FUNCTION_BLOCK fb_palletizeing
VAR_INPUT
END_VAR
VAR_OUTPUT
END_VAR
VAR
	SFCInit: BOOL;
	fbi_coordinateCal: fb_coordinateCal;
	fbi_exchangeTraySystem: fb_exchangeTraySystem;
	trn_pickUpLensDone: BOOL;
	trn_forTray: BOOL;
	trn_forGarbage: BOOL;
	trn_forSample: BOOL;
	trn_trayDone: BOOL;
	trn_garbageDone: BOOL;
	trn_sampleDone: BOOL;
	trn_calculateDone: BOOL;
	var_targetPosX: LREAL;
	var_targetPosY: LREAL;
	var_targetPosZ: LREAL;
	var_process: INT;
	flg_trayIsFull: BOOL;
	flg_sampleIsBusy: BOOL;
	flg_trayIsNotFull: BOOL;
	flg_sampleCavCheck: ARRAY[1..8] OF BOOL;
	var_i: INT;
	flg_bufCavChcek: BOOL;
	trn_moveToInitPosDone: BOOL;
	trn_notTrayChange: BOOL;
	trn_trayChange: BOOL;
	flg_pocketIsNotFull: BOOL;
	trn_trayChangeDone			: BOOL;
	var_cav						: INT;
	trn_DataSamplingDone		: BOOL;
	fbi_vacuumRetry				: fb_vacuumRetry;
	vacuumRetryTimer			: TON;
	var_i_clear					: INT;
	flg_allLensIsNotSet			: BOOL;
	flg_axisSample_Done			: BOOL;
	flg_axisXY_move_Sample_Done	: BOOL;
	fb_TON_delay				: TON;
	fb_TON_delay_error			: TON;
	flg_sample_need				: BOOL;
END_VAR

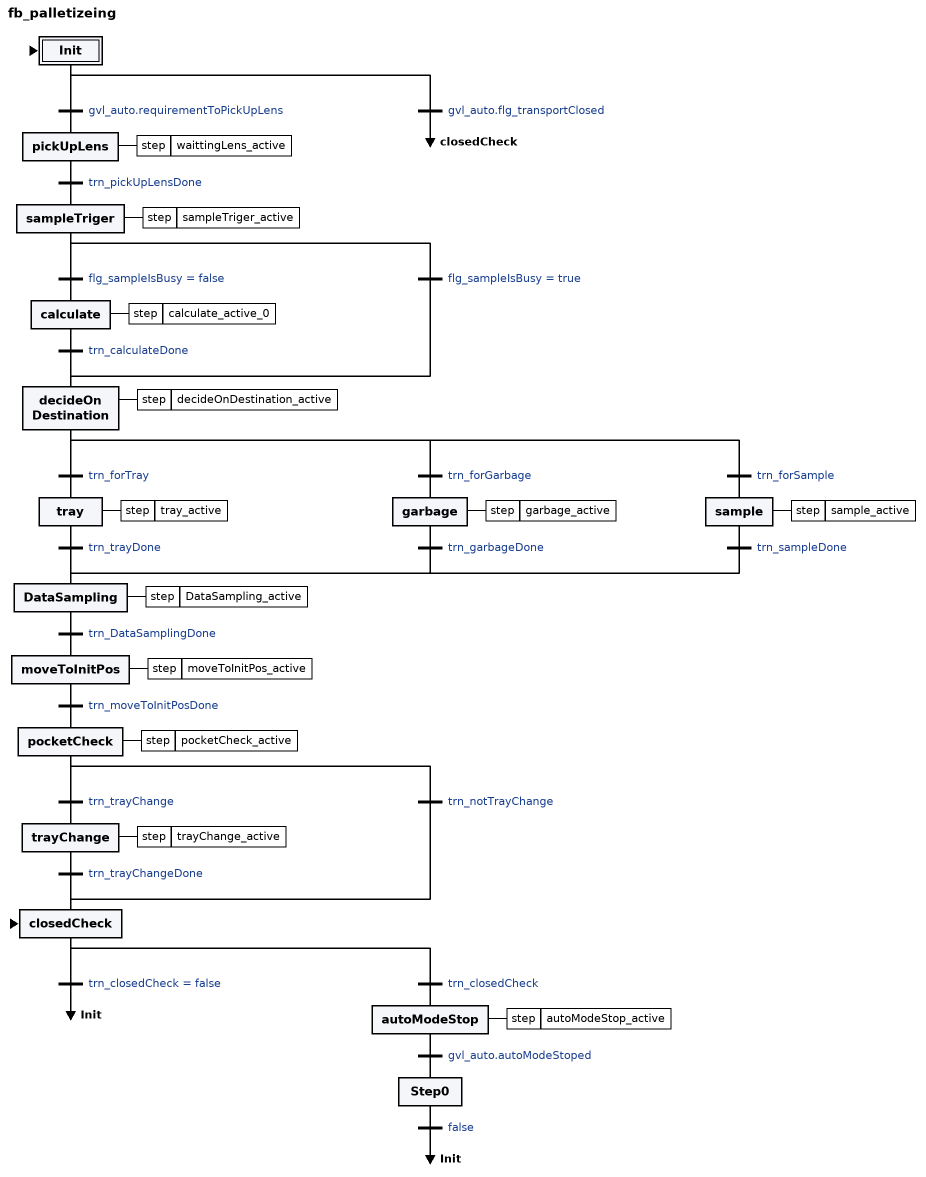
INITIAL_STEP Init:
END_STEP
TRANSITION FROM Init TO pickUpLens
    := gvl_auto.requirementToPickUpLens;
END_TRANSITION
TRANSITION FROM Init TO closedCheck
    := gvl_auto.flg_transportClosed;
END_TRANSITION
STEP pickUpLens:
    waittingLens_active(N);  // step action
END_STEP
TRANSITION FROM pickUpLens TO sampleTriger
    := trn_pickUpLensDone;
END_TRANSITION
STEP sampleTriger:
    sampleTriger_active(N);  // step action
END_STEP
TRANSITION FROM sampleTriger TO calculate
    := flg_sampleIsBusy = false;
END_TRANSITION
STEP calculate:
    calculate_active_0(N);  // step action
END_STEP
TRANSITION FROM calculate TO decideOnDestination
    := trn_calculateDone;
END_TRANSITION
TRANSITION FROM sampleTriger TO decideOnDestination
    := flg_sampleIsBusy = true;
END_TRANSITION
STEP decideOnDestination:
    decideOnDestination_active(N);  // step action
END_STEP
TRANSITION FROM decideOnDestination TO tray
    := trn_forTray;
END_TRANSITION
STEP tray:
    tray_active(N);  // step action
END_STEP
TRANSITION FROM tray TO DataSampling
    := trn_trayDone;
END_TRANSITION
TRANSITION FROM decideOnDestination TO garbage
    := trn_forGarbage;
END_TRANSITION
STEP garbage:
    garbage_active(N);  // step action
END_STEP
TRANSITION FROM garbage TO DataSampling
    := trn_garbageDone;
END_TRANSITION
TRANSITION FROM decideOnDestination TO sample
    := trn_forSample;
END_TRANSITION
STEP sample:
    sample_active(N);  // step action
END_STEP
TRANSITION FROM sample TO DataSampling
    := trn_sampleDone;
END_TRANSITION
STEP DataSampling:
    DataSampling_active(N);  // step action
END_STEP
TRANSITION FROM DataSampling TO moveToInitPos
    := trn_DataSamplingDone;
END_TRANSITION
STEP moveToInitPos:
    moveToInitPos_active(N);  // step action
END_STEP
TRANSITION FROM moveToInitPos TO pocketCheck
    := trn_moveToInitPosDone;
END_TRANSITION
STEP pocketCheck:
    pocketCheck_active(N);  // step action
END_STEP
TRANSITION FROM pocketCheck TO trayChange
    := trn_trayChange;
END_TRANSITION
STEP trayChange:
    trayChange_active(N);  // step action
END_STEP
TRANSITION FROM trayChange TO closedCheck
    := trn_trayChangeDone;
END_TRANSITION
TRANSITION FROM pocketCheck TO closedCheck
    := trn_notTrayChange;
END_TRANSITION
STEP closedCheck:
END_STEP
TRANSITION FROM closedCheck TO Init
    := trn_closedCheck = false;
END_TRANSITION
TRANSITION FROM closedCheck TO autoModeStop
    := trn_closedCheck;
END_TRANSITION
STEP autoModeStop:
    autoModeStop_active(N);  // step action
END_STEP
TRANSITION FROM autoModeStop TO Step0
    := gvl_auto.autoModeStoped;
END_TRANSITION
STEP Step0:
END_STEP
TRANSITION FROM Step0 TO Init
    := false;
END_TRANSITION

ACTION autoModeStop_active:
IF autoModeStop._x AND autoModeStop.x = FALSE THEN
	gvl_auto.autoModeStoped := FALSE;
ELSIF autoModeStop._x AND autoModeStop.x THEN
	gvl_auto.autoModeStoped := TRUE;
END_IF
END_ACTION

ACTION calculate_active_0:
IF calculate._x AND calculate.x = FALSE THEN
	var_process := 0;
	fbi_coordinateCal.in_flg_run := FALSE;
	trn_calculateDone := FALSE;
	flg_trayIsNotFull := FALSE;
ELSIF calculate._x AND calculate.x THEN
	CASE var_process OF
		0:
			var_process := 1;
		1:
			IF  gvl_auto.buf_cavNo <> 0 THEN
				IF  gvl_auto.pocketNo[gvl_auto.buf_cavNo] < gvl_param.var_productInfo[gvl_param.var_currentProductID].pocketSumQty  THEN
					flg_trayIsNotFull := TRUE;
				END_IF
				var_process := 2;
			ELSE
				var_process := 3;
			END_IF
		2:
			fbi_coordinateCal.in_flg_run := TRUE;
			IF fbi_coordinateCal.out_flg_Done THEN
				fbi_coordinateCal.in_flg_run := FALSE;
				var_process := 3;
			END_IF
		3:
			trn_calculateDone := TRUE;
			
	END_CASE
END_IF
fbi_coordinateCal(
	in_flg_run:= , 
	out_flg_run=> , 
	var_ref_productInfo:= gvl_param.var_productInfo[gvl_param.var_currentProductID], 
	in_var_cavNo:= gvl_auto.buf_cavNo, 
	in_var_pocketNo:= gvl_auto.pocketNo[gvl_auto.buf_cavNo] + 1, 
	in_var_calculateMode:= eP_calculateMode.Affine, 
	out_flg_busy=> , 
	out_flg_Done=> , 
	out_var_X=> var_targetPosX, 
	out_var_Y=> var_targetPosY, 
	out_var_Z=> var_targetPosZ);
END_ACTION

ACTION DataSampling_active:
IF DataSampling._x AND DataSampling.x = FALSE THEN
	gvl_auto.flg_dataSampling_run := FALSE;
	trn_DataSamplingDone := FALSE;
ELSIF DataSampling._x AND DataSampling.x THEN
	gvl_auto.flg_dataSampling_run := TRUE;
	trn_DataSamplingDone := TRUE;
END_IF
END_ACTION

ACTION decideOnDestination_active:
IF decideOnDestination._x AND decideOnDestination.x = FALSE THEN
	trn_forTray := FALSE;
	trn_forGarbage := FALSE;
	trn_forSample := FALSE;
	gvl_auto.flg_DataSample_nonDefective := FALSE;
	gvl_auto.flg_DataSample_defective := FALSE;
	gvl_auto.flg_DataSamle_sample := FALSE;
	IF gvl_auto.flg_pocketCountCheck THEN
		gvl_auto.pocketNo[gvl_auto.flg_pocketCountCheck_cav] := gvl_auto.pocketNo[gvl_auto.flg_pocketCountCheck_cav] -1;
	END_IF
ELSIF decideOnDestination._x AND decideOnDestination.x THEN
	gvl_auto.flg_pocketCountCheck_cav := gvl_auto.buf_cavNo;
	gvl_auto.flg_axisIsPcikingUp := FALSE;
	IF flg_trayIsNotFull AND gvl_auto.flg_gateLength AND gvl_auto.buf_cavNo <> 0 AND NOT flg_sampleIsBusy THEN
	//tray
		gvl_auto.flg_pocketCountCheck := TRUE;
		trn_forTray := TRUE;
		gvl_auto.flg_DataSample_nonDefective := TRUE;
	ELSIF flg_sampleIsBusy AND flg_sample_need THEN
	//sample
		gvl_auto.flg_pocketCountCheck := TRUE;
		trn_forSample := TRUE;
		gvl_auto.flg_DataSamle_sample := TRUE;
	ELSE
	//garbage
		IF NOT gvl_auto.flg_gm_eleIsDown THEN
			trn_forGarbage := TRUE;
			gvl_auto.flg_DataSample_defective := TRUE;
		END_IF
	END_IF
END_IF
END_ACTION

ACTION garbage_active:
IF garbage._x AND garbage.x = FALSE THEN
	gvl_axis.fbi_motionControler.in_flg_start := FALSE;
	gvl_solv.fbi_ejector.in_flg_run := FALSE;
	trn_garbageDone := FALSE;
	var_process := 0;
	gvl_auto.var_defectiveLens[gvl_auto.buf_cavNo] := gvl_auto.var_defectiveLens[gvl_auto.buf_cavNo] + 1;
ELSIF garbage._x AND garbage.x THEN
	CASE var_process OF
//		-2:
//			gvl_elecylinder.fbi_axisSample.in_flg_run := FALSE;
//			gvl_elecylinder.fbi_axisSample.in_var_moveMode := eP_eleMoveMode.eleA;
//			gvl_axis.fbi_motionControler.in_flg_start := FALSE;
//			IF gvl_io.flg_frontSaftyDoor THEN
//				gvl_elecylinder.fbi_axisSample.in_flg_run := TRUE;
//				var_process := -1;
//			END_IF
//		-1:
//			IF gvl_elecylinder.fbi_axisSample.out_flg_Done THEN
//				gvl_elecylinder.fbi_axisSample.in_flg_run := FALSE;
//				var_process := 0;
//			END_IF
		0:
			gvl_axis.fbi_motionControler.in_var_targetPosX := gvl_param.var_productInfo[gvl_param.var_currentProductID].teachPos.remove.x;
			gvl_axis.fbi_motionControler.in_var_targetPosY := gvl_param.var_productInfo[gvl_param.var_currentProductID].teachPos.remove.y;
			gvl_axis.fbi_motionControler.in_var_targetPosZ := gvl_param.var_productInfo[gvl_param.var_currentProductID].teachPos.remove.z;
			gvl_axis.fbi_motionControler.in_var_direction := eP_motionDirection.Y_X_Z;
			var_process := 1;
		1:
			gvl_axis.fbi_motionControler.in_flg_start := TRUE;
			var_process := 2;
		2:
			
			IF gvl_axis.fbi_motionControler.out_flg_Done THEN
				gvl_axis.fbi_motionControler.in_flg_start := FALSE;
				var_process := 3;
			END_IF
		3:
			gvl_solv.fbi_ejector.in_var_vacMode := eP_ejeVacMode.break;
			gvl_solv.fbi_ejector.in_flg_run := TRUE;
			var_process := 4;
		4:
			IF gvl_solv.fbi_ejector.out_flg_Done THEN
				gvl_solv.fbi_ejector.in_flg_run := FALSE;
				var_process := 5;
			END_IF
		5:
			gvl_axis.fbi_motionControler.in_flg_start := FALSE;
			gvl_axis.fbi_motionControler.in_var_targetPosX := gvl_param.var_productInfo[gvl_param.var_currentProductID].teachPos.initial.x;
			gvl_axis.fbi_motionControler.in_var_targetPosY := gvl_param.var_productInfo[gvl_param.var_currentProductID].teachPos.remove.y;
			gvl_axis.fbi_motionControler.in_var_targetPosZ := gvl_param.var_productInfo[gvl_param.var_currentProductID].teachPos.initial.z;
			gvl_axis.fbi_motionControler.in_var_direction := eP_motionDirection.Z_X_Y;
			var_process := 6;
		6:
			gvl_axis.fbi_motionControler.in_flg_start := TRUE;
			var_process := 7;
		7:
			
			IF gvl_axis.fbi_motionControler.out_flg_Done THEN
				gvl_axis.fbi_motionControler.in_flg_start := FALSE;
				var_process := 8;
			END_IF
		8:
			gvl_auto.flg_pocketCountCheck := FALSE;
			trn_garbageDone := TRUE;
	END_CASE
END_IF
END_ACTION

ACTION moveToInitPos_active:
IF moveToInitPos._x AND moveToInitPos.x = FALSE THEN
	trn_moveToInitPosDone := FALSE;
	var_process := 0;
ELSIF moveToInitPos._x AND moveToInitPos.x THEN
	CASE var_process OF
		0:
			gvl_axis.fbi_motionControler.in_var_targetPosX := gvl_param.var_productInfo[gvl_param.var_currentProductID].teachPos.initial.x;
			gvl_axis.fbi_motionControler.in_var_targetPosY := gvl_param.var_productInfo[gvl_param.var_currentProductID].teachPos.initial.y;
			gvl_axis.fbi_motionControler.in_var_targetPosZ := gvl_param.var_productInfo[gvl_param.var_currentProductID].teachPos.initial.z;
			gvl_axis.fbi_motionControler.in_var_direction := eP_motionDirection.ZYX;
			var_process := 1;
		1:
			gvl_axis.fbi_motionControler.in_flg_start := TRUE;
			IF gvl_axis.fbi_motionControler.out_flg_Done THEN
				gvl_auto.flg_axisIsPcikingUp := FALSE;
				gvl_axis.fbi_motionControler.in_flg_start := FALSE;
				var_process := 2;
			END_IF
		2:
			gvl_auto.flg_sampling := FALSE;
			trn_moveToInitPosDone := TRUE;
	END_CASE
END_IF
END_ACTION

PROPERTY p_Init : bool
GET
p_init := THIS^.SFCInit;
END_GET
SET
THIS^.SFCInit := p_init;
END_SET
END_PROPERTY

ACTION pocketCheck_active:
IF pocketCheck._x AND pocketCheck.x = FALSE THEN
	trn_trayChange := FALSE;
	trn_notTrayChange := FALSE;
	flg_pocketIsNotFull := FALSE;
ELSIF pocketCheck._x AND pocketCheck.x THEN
	FOR var_i := 1 TO gvl_param.var_productInfo[gvl_param.var_currentProductID].cavQty BY 1 DO
		IF gvl_auto.pocketNo[var_i] < gvl_param.var_productInfo[gvl_param.var_currentProductID].pocketSumQty THEN
			flg_pocketIsNotFull := TRUE;
		END_IF
		IF var_i = gvl_param.var_productInfo[gvl_param.var_currentProductID].cavQty THEN
			trn_trayChange := NOT flg_pocketIsNotFull;
			trn_notTrayChange := flg_pocketIsNotFull;
		END_IF
	END_FOR
END_IF
END_ACTION

ACTION sample_active:
IF sample._x AND sample.x = FALSE THEN
	gvl_axis.fbi_motionControler.in_flg_start := FALSE;
	gvl_elecylinder.fbi_axisSample.in_flg_run := FALSE;
	gvl_error.flg_sample_windown_warning:= FALSE;
	gvl_solv.fbi_ejector.in_flg_run := FALSE;
	flg_axisXY_move_Sample_Done := FALSE;
	flg_axisSample_Done := FALSE;
	trn_sampleDone := FALSE;
	flg_allLensIsNotSet := FALSE;
	gvl_auto.flg_sampling := TRUE;
	fb_TON_delay.IN := FALSE;
	fb_TON_delay_error.IN:= FALSE;
	var_process := -1;
ELSIF sample._x AND sample.x THEN
	fb_TON_delay();
	fb_TON_delay_error(PT:=T#60S);
	CASE var_process OF
		-1:
			var_process:= 0;
		0:
			fb_TON_delay.PT:= T#5S;
			fb_TON_delay.IN:= TRUE;
			fb_TON_delay_error.IN:= TRUE;;
			flg_sampleCavCheck[gvl_auto.buf_cavNo] := TRUE;
			gvl_axis.fbi_motionControler.in_var_targetPosX := gvl_param.var_productInfo[gvl_param.var_currentProductID].teachPos.sample[gvl_auto.buf_cavNo].x;
			gvl_axis.fbi_motionControler.in_var_targetPosY := gvl_param.var_productInfo[gvl_param.var_currentProductID].teachPos.sample[gvl_auto.buf_cavNo].y;
			gvl_axis.fbi_motionControler.in_var_targetPosZ := gvl_param.var_productInfo[gvl_param.var_currentProductID].teachPos.initial.z;
			gvl_axis.fbi_motionControler.in_var_direction := eP_motionDirection.Y_X_Z;
			gvl_elecylinder.fbi_axisSample.in_var_moveMode := eP_eleMoveMode.eleB;
			IF fb_TON_delay.Q THEN
				gvl_error.flg_sample_windown_warning:= TRUE;
				gvl_visu.var_msg:="サンプル台が移動する為に扉を閉じてください。";
			END_IF
			IF fb_TON_delay_error.Q THEN
				gvl_error.flg_sample_windown_error:= TRUE;
				gvl_visu.var_msg:="扉が閉まらないでサンプル台が移動出来ないエラー";
			END_IF
			IF gvl_io.flg_frontSaftyDoor OR gvl_elecylinder.ref_axis_sample.input.in_flg_sensB THEN
				gvl_elecylinder.fbi_axisSample.in_flg_run := TRUE;
				gvl_axis.fbi_motionControler.in_flg_start := TRUE;
				gvl_error.flg_sample_windown_warning:= FALSE;
				fb_TON_delay_error.IN:= FALSE;
				fb_TON_delay.IN := FALSE;
				var_process := 1;
			END_IF
		1:
			IF gvl_elecylinder.fbi_axisSample.out_flg_Done THEN
				flg_axisSample_Done:= TRUE;
				gvl_elecylinder.fbi_axisSample.in_flg_run := FALSE;
			END_IF
			IF gvl_axis.fbi_motionControler.out_flg_Done THEN
				flg_axisXY_move_Sample_Done:= TRUE;
				gvl_axis.fbi_motionControler.in_flg_start := FALSE;
			END_IF
			IF flg_axisSample_Done AND flg_axisXY_move_Sample_Done THEN
				flg_axisSample_Done := FALSE;
				flg_axisXY_move_Sample_Done := FALSE;
				var_process := 2;
			END_IF
		2:
			gvl_axis.fbi_motionControler.in_flg_start := FALSE;
			gvl_axis.fbi_motionControler.in_var_targetPosX := gvl_param.var_productInfo[gvl_param.var_currentProductID].teachPos.sample[gvl_auto.buf_cavNo].X;
			gvl_axis.fbi_motionControler.in_var_targetPosY := gvl_param.var_productInfo[gvl_param.var_currentProductID].teachPos.sample[gvl_auto.buf_cavNo].y;
			gvl_axis.fbi_motionControler.in_var_targetPosZ := gvl_param.var_productInfo[gvl_param.var_currentProductID].teachPos.sample[gvl_auto.buf_cavNo].Z;
			gvl_axis.fbi_motionControler.in_var_direction := eP_motionDirection.Z_X_Y;
			fb_TON_delay.PT:= T#200MS;
			fb_TON_delay.IN:= TRUE;
			IF fb_TON_delay.Q THEN
				fb_TON_delay.IN:= FALSE;
				var_process := 3;
			END_IF
		3:
			gvl_axis.fbi_motionControler.in_flg_start := TRUE;
			var_process := 4;
		4:
			IF gvl_axis.fbi_motionControler.out_flg_Done THEN
				gvl_axis.fbi_motionControler.in_flg_start := FALSE;
				var_process := 5;
			END_IF
		5:
			gvl_solv.fbi_ejector.in_var_vacMode := eP_ejeVacMode.break;
			gvl_solv.fbi_ejector.in_flg_run := TRUE;
			var_process := 6;
		6:
			
			IF gvl_solv.fbi_ejector.out_flg_Done THEN
				gvl_solv.fbi_ejector.in_flg_run := FALSE;
				var_process := 7;
			END_IF	
		7:
			gvl_axis.fbi_motionControler.in_flg_start := FALSE;
			gvl_axis.fbi_motionControler.in_var_targetPosX := gvl_param.var_productInfo[gvl_param.var_currentProductID].teachPos.initial.x;
			gvl_axis.fbi_motionControler.in_var_targetPosY := gvl_param.var_productInfo[gvl_param.var_currentProductID].teachPos.sample[gvl_auto.buf_cavNo].y;
			gvl_axis.fbi_motionControler.in_var_targetPosZ := gvl_param.var_productInfo[gvl_param.var_currentProductID].teachPos.initial.z;
			gvl_axis.fbi_motionControler.in_var_direction := eP_motionDirection.Z_X_Y;
			var_process := 8;
		8:
			gvl_axis.fbi_motionControler.in_flg_start := TRUE;
			var_process := 9;
		9:
			
			IF gvl_axis.fbi_motionControler.out_flg_Done THEN
				gvl_axis.fbi_motionControler.in_flg_start := FALSE;
				var_process := 10;
			END_IF
		10:
			FOR var_i := 1 TO gvl_param.var_productInfo[gvl_param.var_currentProductID].cavQty BY 1 DO
				IF flg_sampleCavCheck[var_i] = FALSE THEN
					flg_allLensIsNotSet := TRUE;
				END_IF
				IF var_i = gvl_param.var_productInfo[gvl_param.var_currentProductID].cavQty THEN
					IF flg_allLensIsNotSet  = FALSE THEN
						flg_sampleIsBusy := FALSE;
						gvl_visu.flg_btn_sample := FALSE;
						var_process := 11;
					ELSE
						var_process := 20;
					END_IF
				END_IF
			END_FOR
		11:
			FOR var_i_clear := 1 TO gvl_param.var_productInfo[gvl_param.var_currentProductID].cavQty BY 1 DO
				flg_sampleCavCheck[var_i_clear] := FALSE;
				IF var_i_clear = gvl_param.var_productInfo[gvl_param.var_currentProductID].cavQty THEN
					var_process := 12;
				END_IF
			END_FOR
		12:
			fb_TON_delay.PT:= T#5S;
			fb_TON_delay.IN:= TRUE;
			fb_TON_delay_error.IN:= TRUE;
			flg_axisSample_Done := FALSE;
			flg_axisXY_move_Sample_Done := FALSE;
			gvl_elecylinder.fbi_axisSample.in_flg_run := FALSE;
			gvl_elecylinder.fbi_axisSample.in_var_moveMode := eP_eleMoveMode.eleA;
			gvl_axis.fbi_motionControler.in_flg_start := FALSE;
			gvl_axis.fbi_motionControler.in_var_targetPosX := gvl_param.var_productInfo[gvl_param.var_currentProductID].teachPos.initial.x;
			gvl_axis.fbi_motionControler.in_var_targetPosY := gvl_param.var_productInfo[gvl_param.var_currentProductID].teachPos.initial.y;
			gvl_axis.fbi_motionControler.in_var_targetPosZ := gvl_param.var_productInfo[gvl_param.var_currentProductID].teachPos.initial.z;
			gvl_axis.fbi_motionControler.in_var_direction := eP_motionDirection.Z_X_Y;
			IF fb_TON_delay.Q THEN
				gvl_error.flg_sample_windown_warning:= TRUE;
				gvl_visu.var_msg:="サンプル台が移動する為に扉を閉じてください。";
			END_IF
			IF fb_TON_delay_error.Q THEN
				gvl_error.flg_sample_windown_error:= TRUE;
				gvl_visu.var_msg:="扉が閉まらないでサンプル台が移動出来ないエラー";
			END_IF
			IF gvl_io.flg_frontSaftyDoor THEN
				gvl_elecylinder.fbi_axisSample.in_flg_run := TRUE;
				gvl_axis.fbi_motionControler.in_flg_start := TRUE;
				gvl_error.flg_sample_windown_warning:= FALSE;
				fb_TON_delay_error.IN:= FALSE;
				fb_TON_delay.IN := FALSE;
				var_process := 13;
			END_IF
		13:
			IF gvl_elecylinder.fbi_axisSample.out_flg_Done THEN
				flg_axisSample_Done:= TRUE;
				gvl_elecylinder.fbi_axisSample.in_flg_run := FALSE;
			END_IF
			IF gvl_axis.fbi_motionControler.out_flg_Done THEN
				flg_axisXY_move_Sample_Done:= TRUE;
				gvl_axis.fbi_motionControler.in_flg_start := FALSE;
			END_IF
			IF flg_axisSample_Done AND flg_axisXY_move_Sample_Done THEN
				flg_axisSample_Done := FALSE;
				flg_axisXY_move_Sample_Done := FALSE;
				var_process := 20;
			END_IF
		20:
			gvl_auto.flg_pocketCountCheck := FALSE;
			trn_sampleDone := TRUE;
	END_CASE
END_IF
END_ACTION

ACTION sampleTriger_active:
IF sampleTriger._x AND sampleTriger.x = FALSE THEN
	IF gvl_visu.flg_btn_sample AND gvl_param.var_productInfo[gvl_param.var_currentProductID].startCav = gvl_auto.buf_cavNo OR flg_sampleIsBusy THEN
		IF flg_sampleCavCheck[gvl_auto.buf_cavNo] THEN
			flg_sample_need := FALSE;
		END_IF
		flg_sampleIsBusy := TRUE;
	ELSE
		flg_sampleIsBusy := FALSE;
	END_IF
ELSIF sampleTriger._x AND sampleTriger.x THEN
	IF gvl_visu.flg_btn_sample AND gvl_param.var_productInfo[gvl_param.var_currentProductID].startCav = gvl_auto.buf_cavNo OR flg_sampleIsBusy THEN
		IF flg_sampleCavCheck[gvl_auto.buf_cavNo] THEN
			flg_sample_need := FALSE;
		END_IF
		flg_sampleIsBusy := TRUE;
	ELSE
		flg_sampleIsBusy := FALSE;
	END_IF
END_IF
END_ACTION

ACTION tray_active:
IF tray._x AND tray.x = FALSE THEN
	gvl_axis.fbi_motionControler.in_flg_start := FALSE;
	gvl_solv.fbi_ejector.in_flg_run := FALSE;
	trn_trayDone := FALSE;
	var_process := 0;
ELSIF tray._x AND tray.x THEN
	IF gvl_visu.var_dev_palletizingMode = FALSE THEN
			CASE var_process OF
				0:
					gvl_axis.fbi_motionControler.in_var_targetPosX := var_targetPosX;
					gvl_axis.fbi_motionControler.in_var_targetPosY := var_targetPosY;
					gvl_axis.fbi_motionControler.in_var_targetPosZ := var_targetPosZ;
					gvl_axis.fbi_motionControler.in_var_direction := eP_motionDirection.XYZ;
					var_process := 1;
				1:
					gvl_axis.fbi_motionControler.in_flg_start := TRUE;
					var_process := 2;
				2:

					IF gvl_axis.fbi_motionControler.out_flg_Done THEN
						gvl_axis.fbi_motionControler.in_flg_start := FALSE;
						var_process := 3;
					END_IF
					//vacuum error check
					IF gvl_axis.fbi_motionControler.out_flg_moveXYDone THEN
						gvl_error.flg_vacuum := NOT gvl_solv.ref_ejector.input.in_flg_sensVac;
					END_IF
				3:
					gvl_solv.fbi_ejector.in_var_vacMode := eP_ejeVacMode.break;
					gvl_auto.pocketNo[gvl_auto.buf_cavNo] := gvl_auto.pocketNo[gvl_auto.buf_cavNo] + 1;
					gvl_solv.fbi_ejector.in_flg_run := TRUE;
					var_process := 4;
				4:
					
					IF gvl_solv.fbi_ejector.out_flg_Done THEN
						gvl_solv.fbi_ejector.in_flg_run := FALSE;
						var_process := 5;
					END_IF
				5:
					gvl_auto.flg_pocketCountCheck := FALSE;
					trn_trayDone := TRUE;
			END_CASE
	ELSIF gvl_visu.var_dev_palletizingMode := TRUE THEN
			CASE var_process OF
				0:
					gvl_axis.fbi_motionControler.in_var_targetPosX := var_targetPosX + gvl_param.var_productInfo[gvl_param.var_currentProductID].teachPos.palletize.upperLower[gvl_param.var_currentTrayPos].cav[gvl_auto.buf_cavNo].teachingDetail.passingPos.x;
					gvl_axis.fbi_motionControler.in_var_targetPosY := var_targetPosY + gvl_param.var_productInfo[gvl_param.var_currentProductID].teachPos.palletize.upperLower[gvl_param.var_currentTrayPos].cav[gvl_auto.buf_cavNo].teachingDetail.passingPos.y;
					gvl_axis.fbi_motionControler.in_var_targetPosZ := var_targetPosZ + gvl_param.var_productInfo[gvl_param.var_currentProductID].teachPos.palletize.upperLower[gvl_param.var_currentTrayPos].cav[gvl_auto.buf_cavNo].teachingDetail.passingPos.z;
					gvl_axis.fbi_motionControler.in_var_direction := eP_motionDirection.XYZ;
					var_process := 1;
				1:
					gvl_axis.fbi_motionControler.in_flg_start := TRUE;
					var_process := 2;
				2:
					
					IF gvl_axis.fbi_motionControler.out_flg_Done THEN
						gvl_axis.fbi_motionControler.in_flg_start := FALSE;
						var_process := 3;
					END_IF
					//vacuum error check
					IF gvl_axis.fbi_motionControler.out_flg_moveXYDone THEN
						gvl_error.flg_vacuum := NOT gvl_solv.ref_ejector.input.in_flg_sensVac;
					END_IF
					
				3:
					gvl_axis.ref_x.Velocity := gvl_param.var_productInfo[gvl_param.var_currentProductID].teachPos.palletize.upperLower[gvl_param.var_currentTrayPos].cav[gvl_auto.buf_cavNo].teachingDetailVels.x.vel;
					gvl_axis.ref_y.Velocity := gvl_param.var_productInfo[gvl_param.var_currentProductID].teachPos.palletize.upperLower[gvl_param.var_currentTrayPos].cav[gvl_auto.buf_cavNo].teachingDetailVels.y.vel;
					gvl_axis.ref_z.Velocity := gvl_param.var_productInfo[gvl_param.var_currentProductID].teachPos.palletize.upperLower[gvl_param.var_currentTrayPos].cav[gvl_auto.buf_cavNo].teachingDetailVels.z.vel;
					gvl_axis.ref_x.Position := var_targetPosX + gvl_param.var_productInfo[gvl_param.var_currentProductID].teachPos.palletize.upperLower[gvl_param.var_currentTrayPos].cav[gvl_auto.buf_cavNo].teachingDetail.settingPOs.x;
					gvl_axis.ref_y.Position := var_targetPosY + gvl_param.var_productInfo[gvl_param.var_currentProductID].teachPos.palletize.upperLower[gvl_param.var_currentTrayPos].cav[gvl_auto.buf_cavNo].teachingDetail.settingPOs.y;
					gvl_axis.ref_z.Position := var_targetPosZ + gvl_param.var_productInfo[gvl_param.var_currentProductID].teachPos.palletize.upperLower[gvl_param.var_currentTrayPos].cav[gvl_auto.buf_cavNo].teachingDetail.settingPOs.z;
					var_process := 4;
				4:
					gvl_axis.ref_x.Execute := TRUE;
					gvl_axis.ref_y.Execute := TRUE;
					gvl_axis.ref_z.Execute := TRUE;
					var_process := 5;
			
				5:
					IF gvl_axis.fbi_mc_absX.Done AND gvl_axis.fbi_mc_absY.Done AND gvl_axis.fbi_mc_absZ.Done THEN
						var_process := 6;
					END_IF
				6:
					gvl_axis.ref_x.Execute := FALSE;
					gvl_axis.ref_y.Execute := FALSE;
					gvl_axis.ref_z.Execute := FALSE;
					gvl_solv.fbi_ejector.in_var_vacMode := eP_ejeVacMode.break;
					gvl_auto.pocketNo[gvl_auto.buf_cavNo] := gvl_auto.pocketNo[gvl_auto.buf_cavNo] + 1;
					gvl_solv.fbi_ejector.in_flg_run := TRUE;
					var_process := 7;
				7:
					
					IF gvl_solv.fbi_ejector.out_flg_Done THEN
						gvl_solv.fbi_ejector.in_flg_run := FALSE;
						var_process := 8;
					END_IF
				8:
					gvl_axis.ref_x.Velocity := gvl_param.var_productInfo[gvl_param.var_currentProductID].autoVels.x.vel;
					gvl_axis.ref_y.Velocity := gvl_param.var_productInfo[gvl_param.var_currentProductID].autoVels.y.vel;
					gvl_axis.ref_z.Velocity := gvl_param.var_productInfo[gvl_param.var_currentProductID].autoVels.z.vel;
					gvl_auto.flg_pocketCountCheck := FALSE;
					trn_trayDone := TRUE;
			END_CASE
	END_IF
END_IF
END_ACTION

ACTION trayChange_active:
IF trayChange._x AND trayChange.x = FALSE THEN
	trn_trayChangeDone := FALSE;
	fbi_exchangeTraySystem.in_flg_start := FALSE;
ELSIF trayChange._x AND trayChange.x THEN
	fbi_exchangeTraySystem.in_flg_start := gvl_visu.flg_btn_trayChangeDone;
	trn_trayChangeDone := NOT gvl_visu.flg_btn_trayChangeDone;
	IF gvl_auto.flg_trayChangeDone THEN
		FOR var_i := 0 TO 8 BY 1 DO
			gvl_auto.pocketNo[var_i] := 0;
			IF var_i = 8 THEN
				fbi_exchangeTraySystem.in_flg_start := FALSE;
				gvl_visu.flg_btn_trayChangeDone := FALSE;
				trn_trayChangeDone := TRUE;
			END_IF
		END_FOR
	END_IF
END_IF
fbi_exchangeTraySystem(
	var_ref_ele:= gvl_elecylinder.ref_axis_trayChange, 
	in_flg_run:= TRUE, 
	in_flg_start:= , 
	in_flg_pause:= NOT gvl_io.flg_frontSaftyDoor, 
	out_flg_run=> , 
	out_flg_busy=> , 
	out_flg_Done=> gvl_auto.flg_trayChangeDone, 
	out_flg_error=> );
END_ACTION

TRANSITION trn_closedCheck:
IF gvl_auto.autoModeStop AND gvl_auto.flg_transportClosed THEN
	trn_closedCheck := TRUE;
ELSE
	trn_closedCheck := FALSE;
END_IF
END_TRANSITION

ACTION waittingLens_active:
IF pickUpLens._x AND pickUpLens.x = FALSE THEN
	vacuumRetryTimer.IN := FALSE;
	gvl_auto.flg_VacuumRetry := FALSE;
	gvl_solv.fbi_ejector.in_var_vacMode := eP_ejeVacMode.halt;
	gvl_axis.fbi_motionControler.in_flg_start := FALSE;
	gvl_axis.fbi_motionControler.in_var_targetPosX := gvl_param.var_productInfo[gvl_param.var_currentProductID].teachPos.pickUp.x;
	gvl_axis.fbi_motionControler.in_var_targetPosY := gvl_param.var_productInfo[gvl_param.var_currentProductID].teachPos.pickUp.y;
	gvl_axis.fbi_motionControler.in_var_targetPosZ := gvl_param.var_productInfo[gvl_param.var_currentProductID].teachPos.pickUp.z;
	gvl_axis.fbi_motionControler.in_var_direction := eP_motionDirection.XYZ;
	trn_pickUpLensDone := FALSE;
	gvl_auto.flg_axisIsPcikingUp := FALSE;
	var_process := 0;
	fbi_vacuumRetry.in_flg_run := FALSE;
	gvl_auto.flg_sampling := FALSE;
ELSIF pickUpLens._x AND pickUpLens.x THEN

	CASE var_process OF
		0:
			IF gvl_auto.requirementToPickUpLens THEN
				IF gvl_visu.flg_btn_usingMeasurementSystem THEN
					IF NOT gvl_auto.flg_gm_eleIsDown THEN
						gvl_auto.flg_axisIsPcikingUp := TRUE;
						gvl_axis.fbi_motionControler.in_flg_start := TRUE;
						var_process := 1;
					END_IF
				ELSE
					gvl_axis.fbi_motionControler.in_flg_start := TRUE;
					var_process := 1;
				END_IF
			END_IF
		1:
			IF gvl_axis.fbi_motionControler.out_flg_Done THEN
				gvl_solv.fbi_ejector.in_flg_run := TRUE;
				gvl_axis.fbi_motionControler.in_flg_start := FALSE;
				var_process := 2;
			END_IF
		2:
			vacuumRetryTimer.IN := TRUE;
			IF vacuumRetryTimer.Q THEN
				var_process := 3;
			END_IF
		3:
			gvl_auto.lensVacuumDone := TRUE;
			IF gvl_auto.chuckopenDone THEN
				var_process := 4;
			END_IF
		4:
			gvl_axis.fbi_motionControler.in_flg_start := FALSE;
			gvl_axis.fbi_motionControler.in_var_targetPosX := gvl_param.var_productInfo[gvl_param.var_currentProductID].teachPos.initial.x;
			gvl_axis.fbi_motionControler.in_var_targetPosY := gvl_param.var_productInfo[gvl_param.var_currentProductID].teachPos.initial.y;
			gvl_axis.fbi_motionControler.in_var_targetPosZ := gvl_param.var_productInfo[gvl_param.var_currentProductID].teachPos.initial.z;
			gvl_axis.fbi_motionControler.in_var_direction := eP_motionDirection.ZYX;
			var_process := 5;
		5:
			gvl_axis.fbi_motionControler.in_flg_start := TRUE;
			var_process := 6;
		6:
			
			IF gvl_axis.fbi_motionControler.out_flg_Done THEN
				var_process := 7;
			END_IF
		7:
			IF NOT gvl_solv.ref_ejector.input.in_flg_sensVac THEN
				fbi_vacuumRetry.in_flg_run := TRUE;
				var_process := 8;
			ELSE
				var_process := 20;
			END_IF
		8:
			IF fbi_vacuumRetry.out_flg_Done THEN
				var_process := 20;
			ELSIF fbi_vacuumRetry.out_flg_faied THEN
				var_process := 10;
			END_IF
		10:
					
		20:	
			flg_sample_need:=TRUE;
			gvl_auto.pickUpLnesDone := TRUE;
			trn_pickUpLensDone := TRUE;
		
		END_CASE
END_IF
vacuumRetryTimer(IN:= , PT:=T#0.3S , Q=> , ET=> );
fbi_vacuumRetry(in_flg_run:= , out_flg_faied=> , out_flg_Done=> );
END_ACTION

END_FUNCTION_BLOCK

(* stored: Version 1.1.0.1, ProductVersion 3.1.4024.11
   POU fb_palletizeing: Id {8e1986b9-49ba-4497-8301-2a0faca06868}, SpecialFunc None
   Action autoModeStop_active: Id {8cbabf1a-ace9-480b-9aaa-a7e127bc4d4c}
   Action calculate_active_0: Id {59deca66-0737-483f-9b64-3054d37a9ccc}
   Action DataSampling_active: Id {98bc9bda-8d33-40c1-baab-725c6f9a6ba7}
   Action decideOnDestination_active: Id {cea5b2b2-de3b-4aa6-9171-a84005f08f5e}
   Action garbage_active: Id {2227d6a9-d120-4017-8624-1b0df330311a}
   Action moveToInitPos_active: Id {7f8fee6b-238e-489e-9ba6-3c269521315b}
   Property p_Init: Id {61bb8438-f049-4ba7-991c-7da88a946eb1}
   Get Get: Id {a1182f4e-4770-4917-8079-79c82b649d07}
   Set Set: Id {45f62133-896f-4095-b5f0-91ec6d494074}
   Action pocketCheck_active: Id {8af681dc-325b-488e-9ae4-86534a219986}
   Action sample_active: Id {ec8c2f02-ebd6-4863-8380-097e5f030b8a}
   Action sampleTriger_active: Id {18902de7-3d7b-4e54-97f8-42ea68badb89}
   Action tray_active: Id {08d7a0c0-d241-4660-aeff-fc2ceabe1ae4}
   Action trayChange_active: Id {b10e854e-689f-4156-8eca-e6f2e8c9648e}
   Transition trn_closedCheck: Id {4bc0fda9-0b97-4c9d-b376-b42914a7011b}
   Action waittingLens_active: Id {f1ade98e-8b41-42fa-a21a-765b809ccd55} *)
